{attribute 'GeneratedUsingTerminal: EK1122-0000-0018'}
{attribute addProperty BoxType "EK1122-0000-0018"}
{attribute addProperty Id "Beckhoff_EJ5xxxsub_EK1100EK1100_AB5A94672"}
{attribute addProperty CRC "1175890828"}
{attribute addProperty Size "2"}
TYPE Beckhoff_EJ5xxxEK1122_4616AB8C EXTENDS EK1122_AB5A9467 :
STRUCT
	{attribute addProperty Name "Beckhoff_EJ5xxxsub_EK1100"}
	Beckhoff_EJ5xxxsub_EK1100 : EK1100_AB5A9467;
END_STRUCT
END_TYPE

(* stored: Version 1.2.0.0, ProductVersion 3.1.4024.9
   DUT Beckhoff_EJ5xxxEK1122_4616AB8C: Id {9df06bfa-5c5b-4027-b413-9742e15985b6} *)
